PROGRAM MAIN
VAR
	
END_VAR

//Auto Logging
AutoLogData();

END_PROGRAM

(* stored: Version 1.1.0.1, ProductVersion 3.1.4024.12
   POU MAIN: Id {e55b49cc-834b-4aa1-9443-3cc72152a800}, SpecialFunc None *)
